TYPE ST_PriceInfo :
STRUCT
	current		: ST_Result;
	today		: ARRAY [0..23] OF ST_Result;
	tomorrow	: ARRAY [0..23] OF ST_Result;
END_STRUCT
END_TYPE

(* stored: Version 1.1.0.1, ProductVersion 3.1.4024.11
   DUT ST_PriceInfo: Id {33a11925-bcf7-49ba-8211-6dca925d8841} *)
